// TIA Portal V21 export
VAR_GLOBAL   // PLC tag table "K_TipoSezionePastorizzatore"
END_VAR
VAR_GLOBAL CONSTANT   // user constants
   K_TipoSezionePastorizzatore_Calda : Int := 0;
   K_TipoSezionePastorizzatore_Fredda : Int := 1;
   K_TipoSezionePastorizzatore_Mista : Int := 2;   // Sia calda che fredda
END_VAR
